FUNCTION_BLOCK PUBLIC FB_VALVE_TIMEOUT_ALARM
VAR_IN_OUT
	Handler : FB_ALARM_HANDLER;
	Config : TYP_VALVE_TIMEOUT_ALARM_CONF;
END_VAR
VAR_INPUT
	Condition : BOOL;
END_VAR
VAR_OUTPUT
	Error : BOOL;
END_VAR
VAR
	_alarm : FB_ALARM;
	Timer : TON;
	PosEdge : R_TRIG;
	NegEdge : F_TRIG;
END_VAR

Timer(IN := Condition, PT := Config.Delay);

PosEdge(CLK := Timer.Q);
NegEdge(CLK := Timer.Q);

_alarm(Handler := Handler);

IF PosEdge.Q AND Config.Enable THEN
	_alarm.Activate();
END_IF;

IF NegEdge.Q THEN
	_alarm.Reset();
END_IF;

Error := Timer.Q;

PROPERTY PUBLIC Alarm : REFERENCE TO FB_ALARM
GET
Alarm REF= THIS^._alarm;
END_GET
END_PROPERTY

END_FUNCTION_BLOCK

(* stored: Version 1.1.0.1, ProductVersion 3.1.4024.12
   POU FB_VALVE_TIMEOUT_ALARM: Id {5a1e804e-ce2a-4294-be03-33d8dc9254b6}, SpecialFunc None
   Property Alarm: Id {1e29ebee-bb90-418d-ba9e-85cbc6413840}
   Get Get: Id {16cae72b-e73f-4a9a-b2de-1ea0a390f88b} *)
